// TIA Portal project "FactoryIO_Template_S7-1500_V15" (V15)

(* hardware
DEVICE "S71500/ET200MP-Station_1"  S7-1500 station
   slot 0: "Profilschiene_0"  6ES7 590-1***0-0AA0
   slot 1: "PLC_1"  CPU 1511-1 PN  6ES7 511-1AK00-0AB0  V1.8
   slot 2: "AI 8xU/I/RTD/TC ST_1"  AI 8xU/I/RTD/TC ST  6ES7 531-7KF00-0AB0  V2.0
   slot 3: "AI 8xU/I/RTD/TC ST_2"  AI 8xU/I/RTD/TC ST  6ES7 531-7KF00-0AB0  V2.0
   slot 4: "AI 8xU/I/RTD/TC ST_3"  AI 8xU/I/RTD/TC ST  6ES7 531-7KF00-0AB0  V2.0
   slot 5: "AI 8xU/I/RTD/TC ST_4"  AI 8xU/I/RTD/TC ST  6ES7 531-7KF00-0AB0  V2.0
   slot 6: "DI 16x24VDC BA_1"  DI 16x24VDC BA  6ES7 521-1BH10-0AA0  V1.0
*)

// ===== PLC "PLC_1"  CPU 1511-1 PN =====

VAR_GLOBAL   // PLC tag table "Standard-Variablentabelle"
   "Tag_1" AT %E0.0 : Bool;
   "Tag_2" AT %A0.0 : Bool;
   "Tag_3" AT %E0.1 : Bool;
   "Estado Reposo" AT %M0.0 : Bool;
   "EstadoCajahaciaDer" AT %M0.1 : Bool;
   "EstadoCajaender" AT %M0.2 : Bool;
   "bandaDer" AT %Q10.0 : Bool;
   "bandaizq" AT %Q10.1 : Bool;
   "start" AT %I10.0 : Bool;
   "sensorizq" AT %I10.1 : Bool;
   "sensorder" AT %I10.2 : Bool;
   "estadocajahaciaiqz" AT %M0.3 : Bool;
   "estadocajahaciacentro" AT %M0.4 : Bool;
   "estadocajaencentro" AT %M0.5 : Bool;
   "estadocajaenizq" AT %M0.6 : Bool;
   "sensorcentro" AT %I10.3 : Bool;
END_VAR

// folder: System blocks/Program resources

DATA_BLOCK "IEC_Counter_0_DB"   // DB1
{ S7_Optimized_Access := 'TRUE' }
AUTHOR : Simatic
FAMILY : IEC
NAME : CNTR
VERSION : 1.0
// stored: InstanceOfName IEC_COUNTER
"IEC_COUNTER"
BEGIN
END_DATA_BLOCK

// folder: (top level)

FUNCTION "MHJ-PLC-Lab-Function-S71500" : Void   // FC9000, SCL
{ S7_Optimized_Access := 'TRUE' }
VERSION : 0.1
   VAR_TEMP
      Value : Byte;
      ForCounter : Int;
   END_VAR
   VAR CONSTANT
      Value_01_DW : DWord := 16#1223_5486;
      Value_02_DW : DWord := 16#A6C9_D1F5;
   END_VAR
BEGIN

   #Value:=PEEK(area := 16#82,
        dbNumber := 0,
        byteOffset := 511);
   #Value := #Value + 1;

   POKE(area := 16#82,
        dbNumber := 0,
        byteOffset := 511,
        value := #Value);

   POKE(area := 16#82,
        dbNumber := 0,
        byteOffset := 1016,
        value := #Value_01_DW);
   POKE(area := 16#82,
        dbNumber := 0,
        byteOffset := 1020,
        value := #Value_02_DW);

   FOR #ForCounter := 0 TO 63 DO
       #Value:=PEEK(area := 16#1,
            dbNumber := 0,
            byteOffset := #ForCounter);
       POKE(area := 16#81,
            dbNumber := 0,
            byteOffset := #ForCounter,
            value := #Value);
   END_FOR;
   #Value := PEEK(area := 16#1,
                  dbNumber := 0,
                  byteOffset := 512);
   POKE(area := 16#82,
        dbNumber := 0,
        byteOffset := 512,
        value := #Value);
END_FUNCTION

ORGANIZATION_BLOCK "Main"   // OB1, LAD, ProgramCycle
TITLE = "Main Program Sweep (Cycle)"
{ S7_Optimized_Access := 'TRUE' }
VERSION : 0.1
   VAR_INPUT
      Initial_Call : Bool;   // Initial call of this OB
      Remanence : Bool;   // =True, if remanent data are available
   END_VAR
   VAR_TEMP   // added for the SCL form of the ladder/FBD networks
      _w1 : Bool;
   END_VAR
BEGIN

REGION Network 1
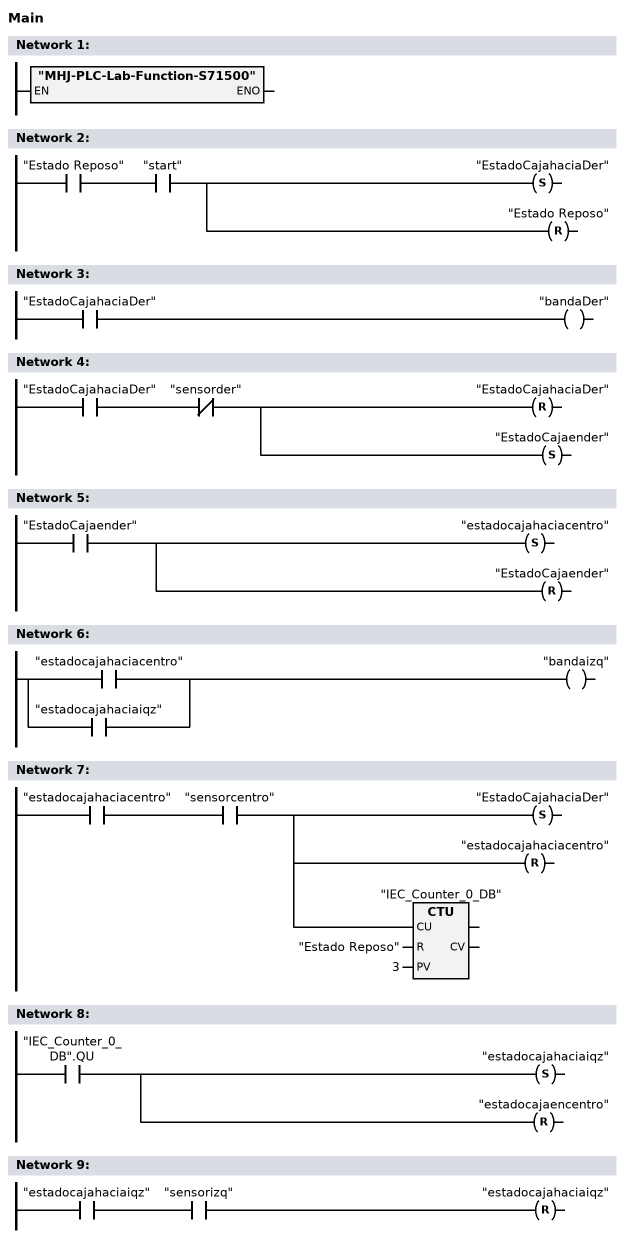
   RUNG wire#powerrail
      "MHJ-PLC-Lab-Function-S71500"()
   END_RUNG
   // the same network as SCL:
   "MHJ-PLC-Lab-Function-S71500"();
END_REGION

REGION Network 2
   RUNG wire#powerrail
      Contact( "Estado Reposo" )
      Contact( "start" )
      wire#w1
      S_Coil( "EstadoCajahaciaDer" )
   END_RUNG
   RUNG wire#w1
      R_Coil( "Estado Reposo" )
   END_RUNG
   // the same network as SCL:
   IF "Estado Reposo" AND "start" THEN
       "EstadoCajahaciaDer" := TRUE;
       "Estado Reposo" := FALSE;
   END_IF;
END_REGION

REGION Network 3
   RUNG wire#powerrail
      Contact( "EstadoCajahaciaDer" )
      Coil( "bandaDer" )
   END_RUNG
   // the same network as SCL:
   "bandaDer" := "EstadoCajahaciaDer";
END_REGION

REGION Network 4
   RUNG wire#powerrail
      Contact( "EstadoCajahaciaDer" )
      I_Contact( "sensorder" )
      wire#w1
      R_Coil( "EstadoCajahaciaDer" )
   END_RUNG
   RUNG wire#w1
      S_Coil( "EstadoCajaender" )
   END_RUNG
   // the same network as SCL:
   #_w1 := "EstadoCajahaciaDer" AND NOT "sensorder";
   IF #_w1 THEN
       "EstadoCajahaciaDer" := FALSE;
       "EstadoCajaender" := TRUE;
   END_IF;
END_REGION

REGION Network 5
   RUNG wire#powerrail
      Contact( "EstadoCajaender" )
      wire#w1
      S_Coil( "estadocajahaciacentro" )
   END_RUNG
   RUNG wire#w1
      R_Coil( "EstadoCajaender" )
   END_RUNG
   // the same network as SCL:
   IF "EstadoCajaender" THEN
       "estadocajahaciacentro" := TRUE;
       "EstadoCajaender" := FALSE;
   END_IF;
END_REGION

REGION Network 6
   RUNG wire#powerrail
      Contact( "estadocajahaciacentro" )
      wire#w1
      Coil( "bandaizq" )
   END_RUNG
   RUNG wire#powerrail
      Contact( "estadocajahaciaiqz" )
   END_RUNG wire#w1
   // the same network as SCL:
   "bandaizq" := "estadocajahaciacentro" OR "estadocajahaciaiqz";
END_REGION

REGION Network 7
   #_w1 := "estadocajahaciacentro" AND "sensorcentro";
   IF #_w1 THEN
       "EstadoCajahaciaDer" := TRUE;
       "estadocajahaciacentro" := FALSE;
   END_IF;
   "IEC_Counter_0_DB".CTU(CU := #_w1, R := "Estado Reposo", PV := 3);
END_REGION

REGION Network 8
   RUNG wire#powerrail
      Contact( "IEC_Counter_0_DB".QU )
      wire#w1
      S_Coil( "estadocajahaciaiqz" )
   END_RUNG
   RUNG wire#w1
      R_Coil( "estadocajaencentro" )
   END_RUNG
   // the same network as SCL:
   IF "IEC_Counter_0_DB".QU THEN
       "estadocajahaciaiqz" := TRUE;
       "estadocajaencentro" := FALSE;
   END_IF;
END_REGION

REGION Network 9
   RUNG wire#powerrail
      Contact( "estadocajahaciaiqz" )
      Contact( "sensorizq" )
      R_Coil( "estadocajahaciaiqz" )
   END_RUNG
   // the same network as SCL:
   IF "estadocajahaciaiqz" AND "sensorizq" THEN "estadocajahaciaiqz" := FALSE; END_IF;
END_REGION
END_ORGANIZATION_BLOCK

ORGANIZATION_BLOCK "Startup"   // OB100, LAD, Startup
TITLE = "Complete Restart"
{ S7_Optimized_Access := 'TRUE' }
VERSION : 0.1
   VAR_INPUT
      LostRetentive : Bool;   // True if retentive data are lost
      LostRTC : Bool;   // True if date and time are lost
   END_VAR
BEGIN

REGION Network 1
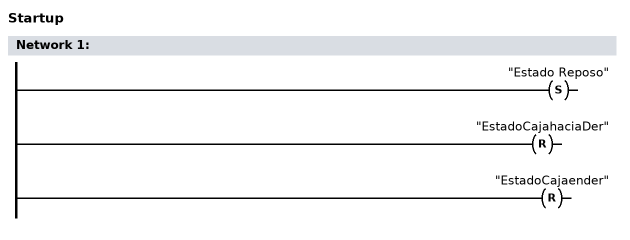
   RUNG wire#powerrail
      S_Coil( "Estado Reposo" )
   END_RUNG
   RUNG wire#powerrail
      R_Coil( "EstadoCajahaciaDer" )
   END_RUNG
   RUNG wire#powerrail
      R_Coil( "EstadoCajaender" )
   END_RUNG
   // the same network as SCL:
   "Estado Reposo" := TRUE;
   "EstadoCajahaciaDer" := FALSE;
   "EstadoCajaender" := FALSE;
END_REGION
END_ORGANIZATION_BLOCK